FUNCTION_BLOCK PUBLIC FB_LampSetDirect IMPLEMENTS I_Subject
VAR
	nLightLevel			:	USINT;
	_ipObserver			:	I_Observer;	
END_VAR

METHOD Attach
VAR_INPUT
	ipObserver		: I_Observer;
END_VAR
IF (ipObserver = 0) THEN
	RETURN;
END_IF
_ipObserver := ipObserver;
END_METHOD

METHOD Detach
_ipObserver := 0;
END_METHOD

// Sets the control value to a value between 0 and 100.
METHOD PUBLIC SetLightLevel
VAR_INPUT
	nNewLightLevel		:	USINT(0..100);
END_VAR
nLightLevel := nNewLightLevel;
IF (_ipObserver <> 0) THEN
	_ipObserver.Update(nLightLevel);
END_IF
END_METHOD

END_FUNCTION_BLOCK

(* stored: Version 1.1.0.1, ProductVersion 3.1.4024.12
   POU FB_LampSetDirect: Id {c9363aa1-33e3-41da-adea-7faeb59d6855}, SpecialFunc None
   Method Attach: Id {7d2c5813-55e6-4687-b48f-e21fdab00ed6}
   Method Detach: Id {d4f7a047-16d7-4520-834a-3ee7d18792e2}
   Method SetLightLevel: Id {4b6fea93-5fee-4ee1-8a77-261782e46dcf} *)
